FUNCTION_BLOCK fb_eje_controller
VAR_IN_OUT
	var_ref_eje : ref_eje_io;
END_VAR
VAR_INPUT
	in_flg_run : BOOL;
	in_var_vacMode : eP_ejeVacMode;
	in_flg_retry: BOOL;
END_VAR
VAR_OUTPUT
	out_flg_run : BOOL;
	out_flg_busy: BOOL;
	out_flg_Done: BOOL;
	out_flg_error : BOOL;
END_VAR
VAR
	var_buf_moveMode: eP_ejeVacMode;
	flg_vacOnDone: BOOL;
	flg_vacOffDone: BOOL;
	flg_vacBreakDone: BOOL;
	flg_vacHaltDone: BOOL;
	fbi_brakTime: TON;
	flg_breakDone: BOOL;
	var_timeOut: TON;
	in: BOOL;
END_VAR
VAR // added by the converter: edge detectors and wires of the graphical bodies
    _rt1, _rt2, _rt3, _rt4 : R_TRIG;
    _w1, _w2, _w3, _w4, _w5 : BOOL;
END_VAR

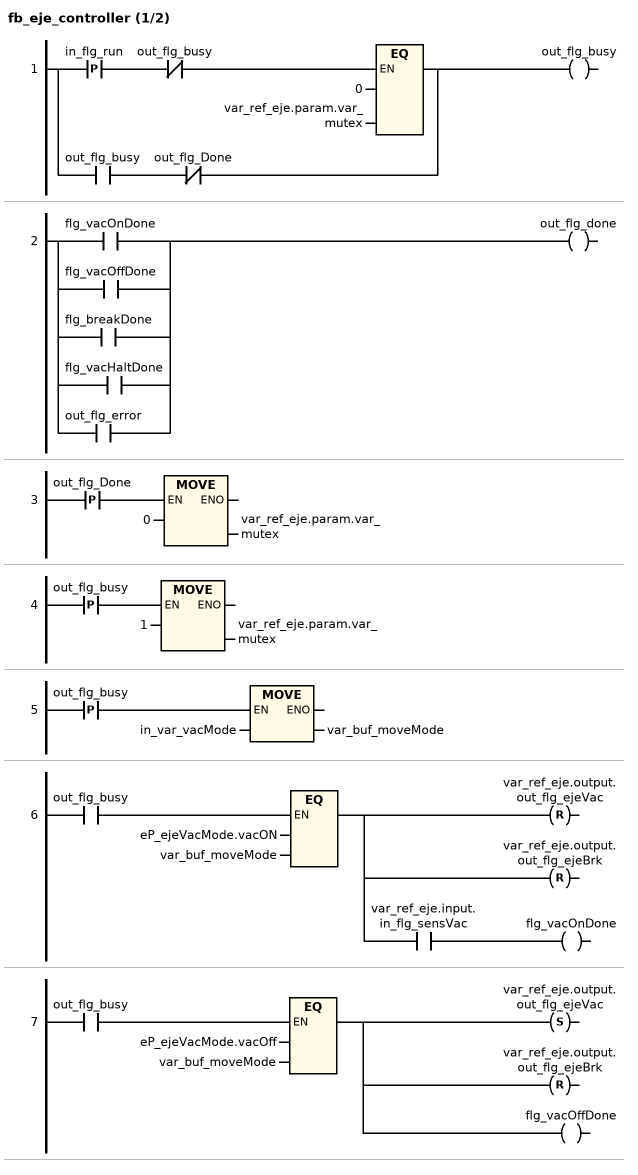
// NETWORK 1
_rt1(CLK := in_flg_run);
out_flg_busy := _rt1.Q AND NOT out_flg_busy AND 0 = var_ref_eje.param.var_mutex OR out_flg_busy AND NOT out_flg_Done;

// NETWORK 2
out_flg_done := flg_vacOnDone OR flg_vacOffDone OR flg_breakDone OR flg_vacHaltDone OR out_flg_error;

// NETWORK 3
_rt2(CLK := out_flg_Done);
IF _rt2.Q THEN var_ref_eje.param.var_mutex := 0; END_IF

// NETWORK 4
_rt3(CLK := out_flg_busy);
IF _rt3.Q THEN var_ref_eje.param.var_mutex := 1; END_IF

// NETWORK 5
_rt4(CLK := out_flg_busy);
IF _rt4.Q THEN var_buf_moveMode := in_var_vacMode; END_IF

// NETWORK 6
_w1 := out_flg_busy AND eP_ejeVacMode.vacON = var_buf_moveMode;
var_ref_eje.output.out_flg_ejeVac R= _w1;
var_ref_eje.output.out_flg_ejeBrk R= _w1;
flg_vacOnDone := _w1 AND var_ref_eje.input.in_flg_sensVac;

// NETWORK 7
_w2 := out_flg_busy AND eP_ejeVacMode.vacOff = var_buf_moveMode;
var_ref_eje.output.out_flg_ejeVac S= _w2;
var_ref_eje.output.out_flg_ejeBrk R= _w2;
flg_vacOffDone := _w2;

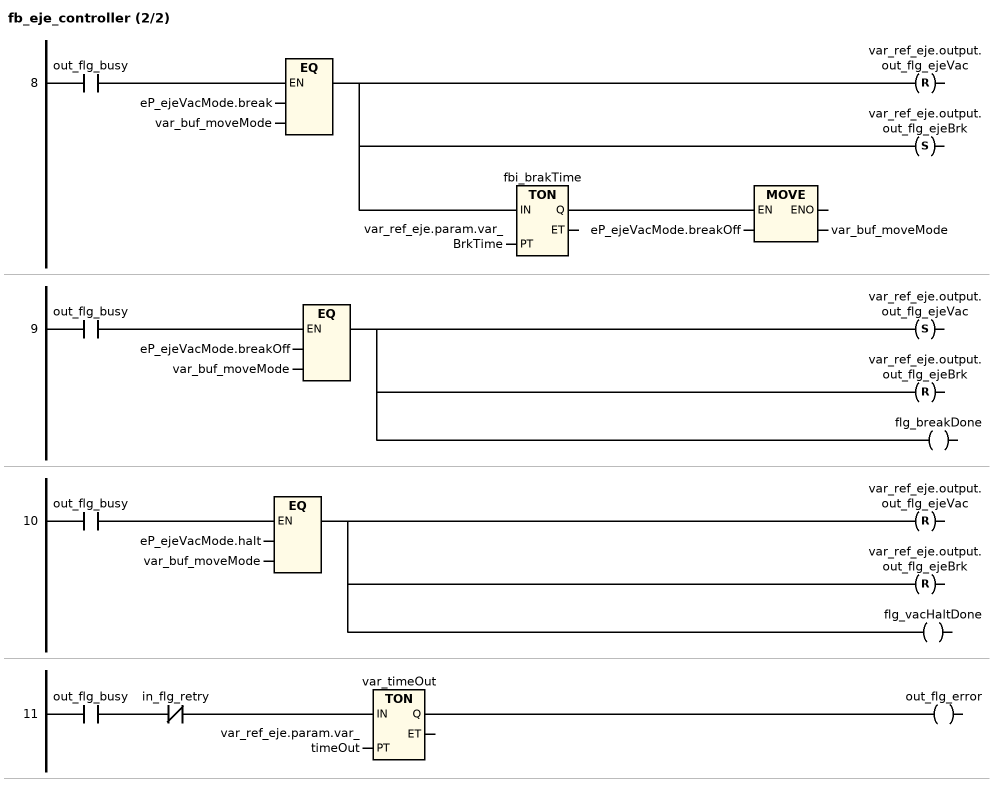
// NETWORK 8
_w3 := out_flg_busy AND eP_ejeVacMode.break = var_buf_moveMode;
var_ref_eje.output.out_flg_ejeVac R= _w3;
var_ref_eje.output.out_flg_ejeBrk S= _w3;
fbi_brakTime(IN := _w3, PT := var_ref_eje.param.var_BrkTime); // TON
IF fbi_brakTime.Q THEN var_buf_moveMode := eP_ejeVacMode.breakOff; END_IF

// NETWORK 9
_w4 := out_flg_busy AND eP_ejeVacMode.breakOff = var_buf_moveMode;
var_ref_eje.output.out_flg_ejeVac S= _w4;
var_ref_eje.output.out_flg_ejeBrk R= _w4;
flg_breakDone := _w4;

// NETWORK 10
_w5 := out_flg_busy AND eP_ejeVacMode.halt = var_buf_moveMode;
var_ref_eje.output.out_flg_ejeVac R= _w5;
var_ref_eje.output.out_flg_ejeBrk R= _w5;
flg_vacHaltDone := _w5;

// NETWORK 11
var_timeOut(IN := out_flg_busy AND NOT in_flg_retry, PT := var_ref_eje.param.var_timeOut); // TON
out_flg_error := var_timeOut.Q;

END_FUNCTION_BLOCK

(* stored: Version 1.1.0.1, ProductVersion 3.1.4024.11
   POU fb_eje_controller: Id {d0b711b4-3e3b-445b-93da-40f91d42d6bb}, SpecialFunc None *)
